PROGRAM MAIN
VAR
	{attribute addProperty Name "Manual"}
	_IsManual : BOOL;
	{attribute addProperty Name "Horizontal piston"}
	horizontalPiston : TcOpen.fbCylinder;
	{attribute addProperty Name "Vertical piston"}
	verticalPiston : TcOpen.fbCylinder;
	{attribute addProperty Name "Gripper piston"}
	gripperPiston : TcOpen.fbCylinder;
END_VAR

IF(_IsManual) THEN
	horizontalPiston.Manual();
	verticalPiston.Manual();
	gripperPiston.Manual();		
END_IF;

END_PROGRAM

(* stored: Version 1.1.0.1, ProductVersion 3.1.4024.4
   POU MAIN: Id {84d391ff-245d-469c-9f07-0280ac5ddd13}, SpecialFunc None *)
